// TIA Portal V18 export
TYPE "UDT_TrackingReport_OP01"
// stored: IsFailsafeCompliant false
   STRUCT
      "Date" : DTL;   // 记录时间
      "P-LineID" : String[18];   // 生产线代号
      "P-StationID" : String[18];   // 工位代号
      "P-PalletNo" : Int;   // 托盘编号
      "P-PalletType" : Byte;   // 托盘类型，1-LOOP1托盘，2-LOOP2托盘等
      "P-PalletStatus" : Byte;   // 预留 托盘状态
      "P-CT_Total" : Real;   // 总循环时间（秒）
      "P-CT_Sub" : Array[1..20] of Real;   // 工步分项节拍时间（秒）
      "P-Data" : "PLCtoMES_OP_ProcessData_OP220";   // 质量终值数据数组
      "P-PartID" : Array[1..10] of String[48];
      "P-SubPartID" : Array[1..10] of String[48];
   END_STRUCT;
END_TYPE
